(* CoDeSys 2.3 export: MonitorBool.EXP *)

(* POU basic/MonitorBool, ST *)
FUNCTION MonitorBool : BOOL
VAR_INPUT
    Value: BOOL;
    Channel: UINT;
END_VAR
VAR_IN_OUT
    Data: BOOL;
END_VAR
VAR
END_VAR
IF Value <> Data THEN
    IF Channel < 256 THEN
        EvtCh8Tick32Bool8(UINT_TO_BYTE(Channel), GlobalTick, Value, GlobalLogBufferHandle);
    ELSE
        EvtCh16Tick32Bool8(Channel, GlobalTick, Value, GlobalLogBufferHandle);
    END_IF
    Data := Value;
END_IF
END_FUNCTION
